// TIA Portal V19 export
TYPE "MachineStatus"
// stored: Access Published
   STRUCT
      AtLeastOneMachineIsAborting { ExternalWritable := 'False'} : Bool;   // One of machine controlled by the area is aborting
      AllMachineAutReady { ExternalWritable := 'False'} : Bool;   // All the machine controlled by the area are Auto ready
      AllMachineAckStopInPhase { ExternalWritable := 'False'} : Bool;   // All the machine controlled by the area return the ack stop in phase
      AllMachineAckStopProgrammed { ExternalWritable := 'False'} : Bool;   // All the machine controlled by the area return the ack stop programmed
      AtLeastOneWngPresence { ExternalWritable := 'False'} : Bool;   // One of machine controlled by the area have a warning
      AtLeastOneAlrPresence { ExternalWritable := 'False'} : Bool;   // One of machine controlled by the area have an alarm
   END_STRUCT;
END_TYPE
